Omron CX-Programmer project NewProject (CX-Programmer 9.73)

# PLC NewPLC1: CP2E-N N

## Global symbols (name address type ; comment)
0.00 BOOL  ; A/M
0.01 BOOL  ; Master On
0.03 BOOL  ; IN
0.04 BOOL  ; OUT
100.00 BOOL  ; AC 1
100.01 BOOL  ; AC 2
100.02 BOOL  ; L4
100.03 BOOL  ; L1
100.04 BOOL  ; L2
100.05 BOOL  ; L3
100.06 BOOL  ; L6
100.07 BOOL  ; L5
101.01 BOOL  ; Buzzer
10.01 BOOL  ; LAMP 4
10.02 BOOL  ; LAMP 1
10.03 BOOL  ; LAMP 2
10.04 BOOL  ; LAMP 3
10.05 BOOL  ; LAMP 6
10.06 BOOL  ; LAMP 5
1.00 BOOL  ; ON_HMI
20.00 BOOL  ; AC1
20.01 BOOL  ; LAMP 4
20.02 BOOL  ; LAMP 1
20.03 BOOL  ; LAMP 2
20.04 BOOL  ; LAMP 3
20.05 BOOL  ; LAMP 6
30.00 BOOL  ; AC 1
30.01 BOOL  ; AC 2
40.00 BOOL  ; AC 1
40.01 BOOL  ; AC 2
60.00 BOOL  ; lampu 1
60.01 BOOL  ; lampu 2
60.02 BOOL  ; lampu 3
60.03 BOOL  ; lampu 4
60.04 BOOL  ; lampu 5
60.05 BOOL  ; lampu 6
60.06 BOOL  ; AC 1
60.07 BOOL  ; AC 2
80.00 BOOL  ; AutoSet
80.01 BOOL  ; Autoful
80.02 BOOL  ; Res
90.00 BOOL  ; AUTO
90.01 BOOL  ; MANUAL
D2.00 BOOL  ; setengah
D300 CHANNEL  ; Error
D500 CHANNEL  ; ]
W60.00 BOOL  ; Setengah
Data1 D600 INT

## Program NewProgram1 (cyclic task 0)
Local symbols
Data UINT
INC BOOL
MOV BOOL
S UINT

### Section MAIN

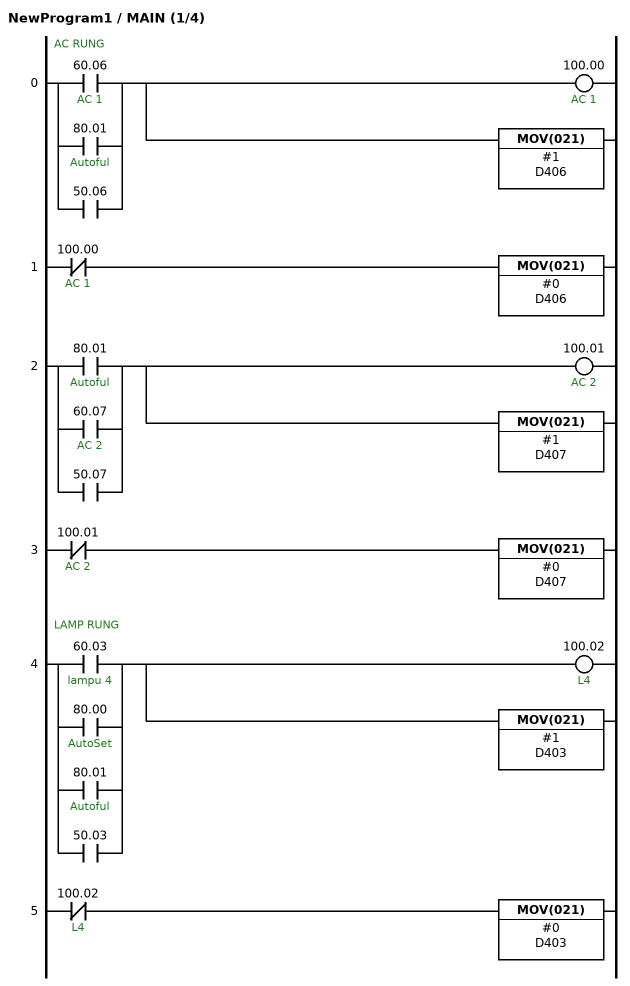
; rung 0: AC RUNG
LD 60.06  ; AC 1
OR 80.01  ; Autoful
OR 50.06
OUT 100.00  ; AC 1
MOV(021) #1 D406
; rung 1
LDNOT 100.00  ; AC 1
MOV(021) #0 D406
; rung 2
LD 80.01  ; Autoful
OR 60.07  ; AC 2
OR 50.07
OUT 100.01  ; AC 2
MOV(021) #1 D407
; rung 3
LDNOT 100.01  ; AC 2
MOV(021) #0 D407
; rung 4: LAMP RUNG
LD 60.03  ; lampu 4
OR 80.00  ; AutoSet
OR 80.01  ; Autoful
OR 50.03
OUT 100.02  ; L4
MOV(021) #1 D403
; rung 5
LDNOT 100.02  ; L4
MOV(021) #0 D403

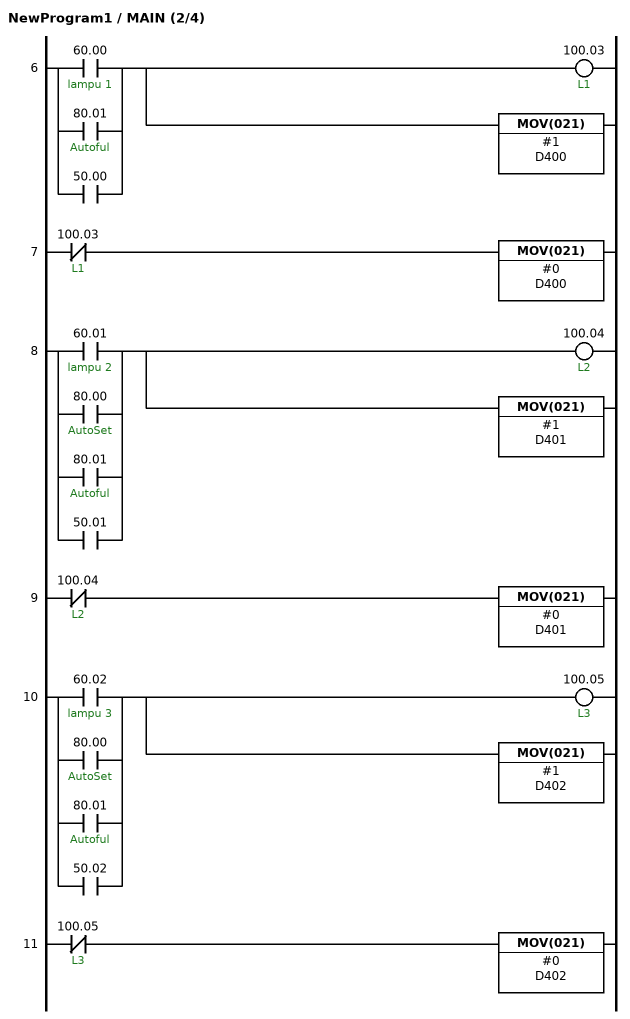
; rung 6
LD 60.00  ; lampu 1
OR 80.01  ; Autoful
OR 50.00
OUT 100.03  ; L1
MOV(021) #1 D400
; rung 7
LDNOT 100.03  ; L1
MOV(021) #0 D400
; rung 8
LD 60.01  ; lampu 2
OR 80.00  ; AutoSet
OR 80.01  ; Autoful
OR 50.01
OUT 100.04  ; L2
MOV(021) #1 D401
; rung 9
LDNOT 100.04  ; L2
MOV(021) #0 D401
; rung 10
LD 60.02  ; lampu 3
OR 80.00  ; AutoSet
OR 80.01  ; Autoful
OR 50.02
OUT 100.05  ; L3
MOV(021) #1 D402
; rung 11
LDNOT 100.05  ; L3
MOV(021) #0 D402

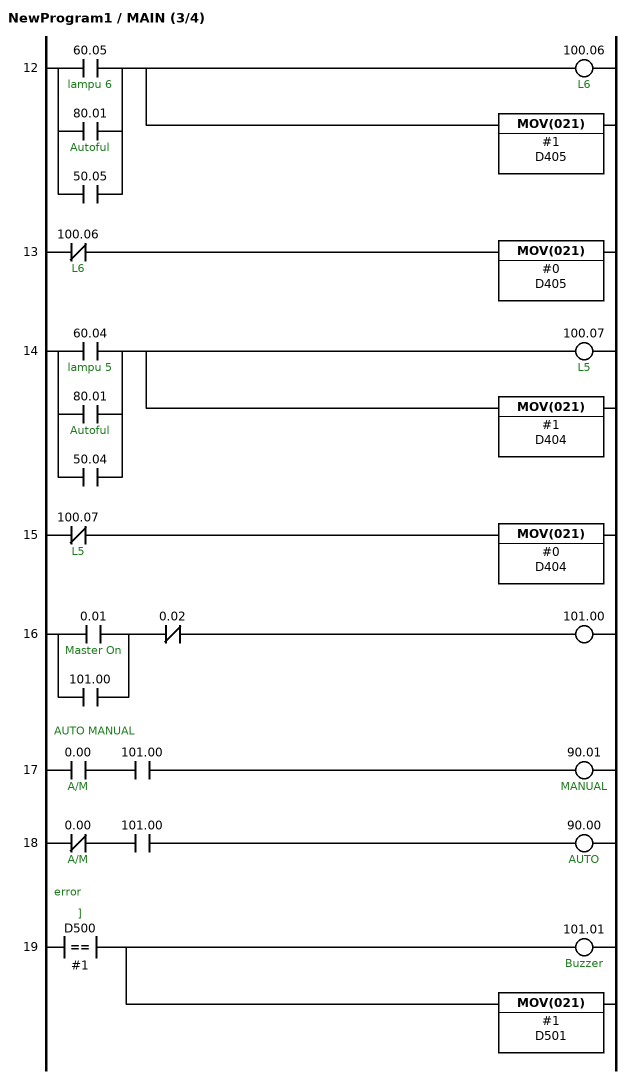
; rung 12
LD 60.05  ; lampu 6
OR 80.01  ; Autoful
OR 50.05
OUT 100.06  ; L6
MOV(021) #1 D405
; rung 13
LDNOT 100.06  ; L6
MOV(021) #0 D405
; rung 14
LD 60.04  ; lampu 5
OR 80.01  ; Autoful
OR 50.04
OUT 100.07  ; L5
MOV(021) #1 D404
; rung 15
LDNOT 100.07  ; L5
MOV(021) #0 D404
; rung 16
LD 0.01  ; Master On
OR 101.00
ANDNOT 0.02
OUT 101.00
; rung 17: AUTO MANUAL
LD 0.00  ; A/M
AND 101.00
OUT 90.01  ; MANUAL
; rung 18
LDNOT 0.00  ; A/M
AND 101.00
OUT 90.00  ; AUTO
; rung 19: error
LD=(300) D500 #1  ; ]
OUT 101.01  ; Buzzer
MOV(021) #1 D501

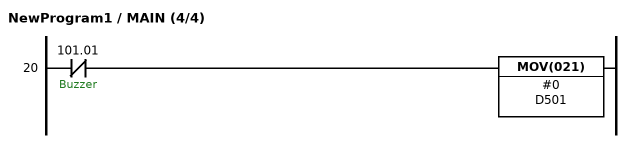
; rung 20
LDNOT 101.01  ; Buzzer
MOV(021) #0 D501

### Section MANUAL___HMI

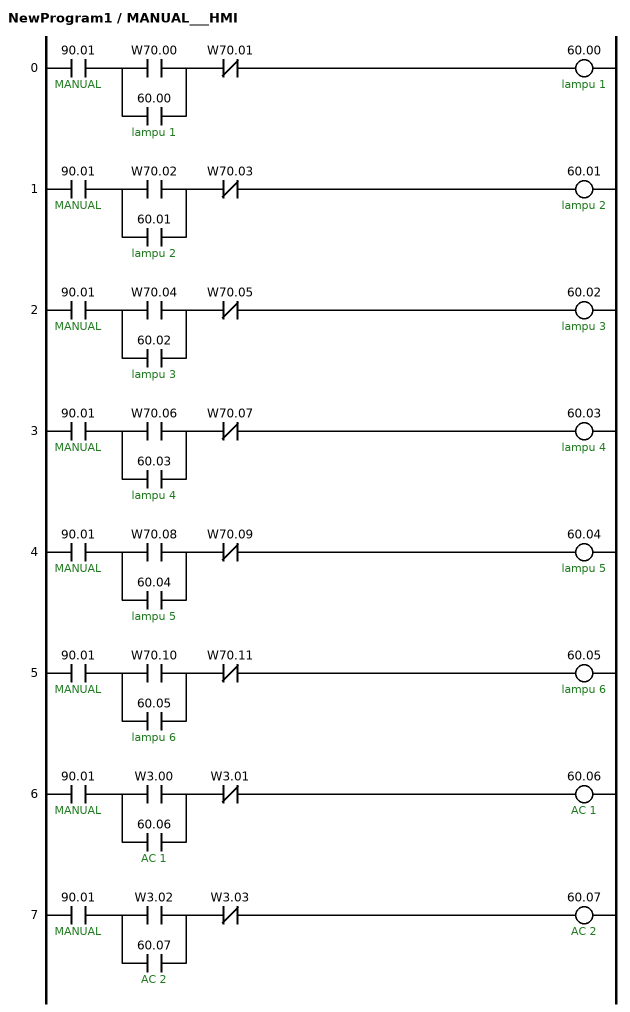
; rung 0
LD 90.01  ; MANUAL
LD W70.00
OR 60.00  ; lampu 1
ANDLD
ANDNOT W70.01
OUT 60.00  ; lampu 1
; rung 1
LD 90.01  ; MANUAL
LD W70.02
OR 60.01  ; lampu 2
ANDLD
ANDNOT W70.03
OUT 60.01  ; lampu 2
; rung 2
LD 90.01  ; MANUAL
LD W70.04
OR 60.02  ; lampu 3
ANDLD
ANDNOT W70.05
OUT 60.02  ; lampu 3
; rung 3
LD 90.01  ; MANUAL
LD W70.06
OR 60.03  ; lampu 4
ANDLD
ANDNOT W70.07
OUT 60.03  ; lampu 4
; rung 4
LD 90.01  ; MANUAL
LD W70.08
OR 60.04  ; lampu 5
ANDLD
ANDNOT W70.09
OUT 60.04  ; lampu 5
; rung 5
LD 90.01  ; MANUAL
LD W70.10
OR 60.05  ; lampu 6
ANDLD
ANDNOT W70.11
OUT 60.05  ; lampu 6
; rung 6
LD 90.01  ; MANUAL
LD W3.00
OR 60.06  ; AC 1
ANDLD
ANDNOT W3.01
OUT 60.06  ; AC 1
; rung 7
LD 90.01  ; MANUAL
LD W3.02
OR 60.07  ; AC 2
ANDLD
ANDNOT W3.03
OUT 60.07  ; AC 2

### Section AUTO

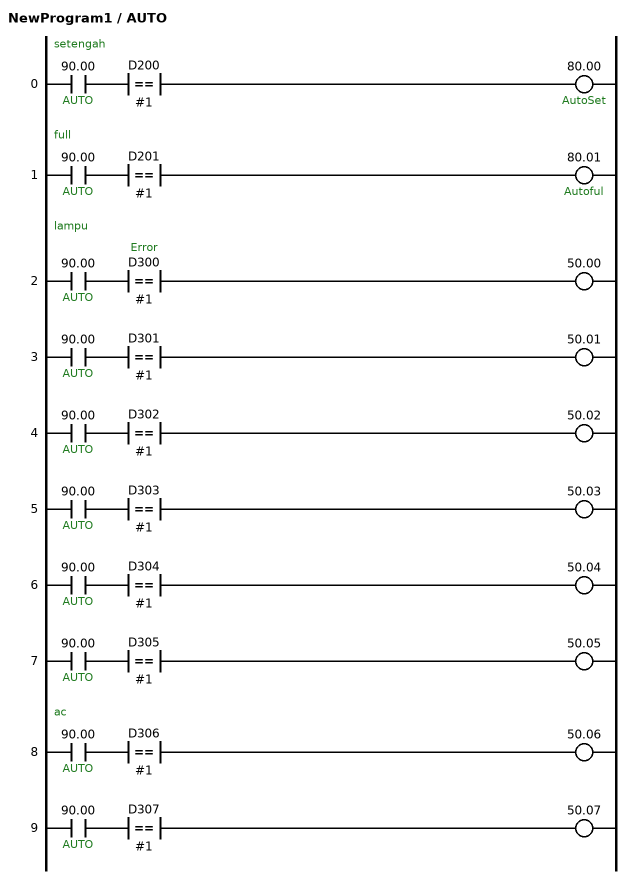
; rung 0: setengah
LD 90.00  ; AUTO
AND=(300) D200 #1
OUT 80.00  ; AutoSet
; rung 1: full
LD 90.00  ; AUTO
AND=(300) D201 #1
OUT 80.01  ; Autoful
; rung 2: lampu
LD 90.00  ; AUTO
AND=(300) D300 #1  ; Error
OUT 50.00
; rung 3
LD 90.00  ; AUTO
AND=(300) D301 #1
OUT 50.01
; rung 4
LD 90.00  ; AUTO
AND=(300) D302 #1
OUT 50.02
; rung 5
LD 90.00  ; AUTO
AND=(300) D303 #1
OUT 50.03
; rung 6
LD 90.00  ; AUTO
AND=(300) D304 #1
OUT 50.04
; rung 7
LD 90.00  ; AUTO
AND=(300) D305 #1
OUT 50.05
; rung 8: ac
LD 90.00  ; AUTO
AND=(300) D306 #1
OUT 50.06
; rung 9
LD 90.00  ; AUTO
AND=(300) D307 #1
OUT 50.07

### Section Simulator

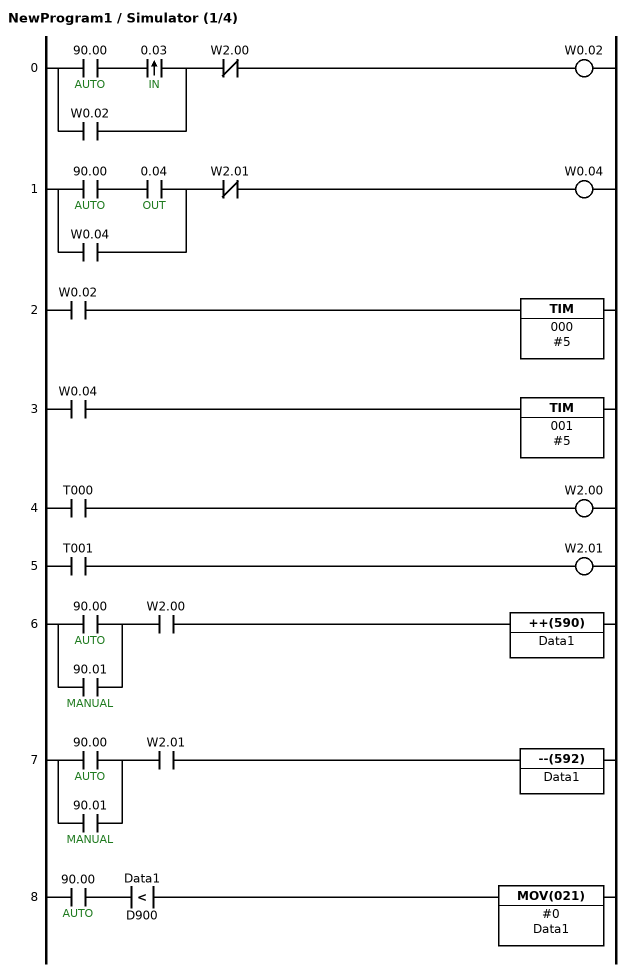
; rung 0
LD 90.00  ; AUTO
@AND 0.03  ; IN
OR W0.02
ANDNOT W2.00
OUT W0.02
; rung 1
LD 90.00  ; AUTO
AND 0.04  ; OUT
OR W0.04
ANDNOT W2.01
OUT W0.04
; rung 2
LD W0.02
TIM 000 #5
; rung 3
LD W0.04
TIM 001 #5
; rung 4
LD T000
OUT W2.00
; rung 5
LD T001
OUT W2.01
; rung 6
LD 90.00  ; AUTO
OR 90.01  ; MANUAL
AND W2.00
++(590) Data1
; rung 7
LD 90.00  ; AUTO
OR 90.01  ; MANUAL
AND W2.01
--(592) Data1
; rung 8
LD 90.00  ; AUTO
AND<S(312) Data1 D900
MOV(021) #0 Data1

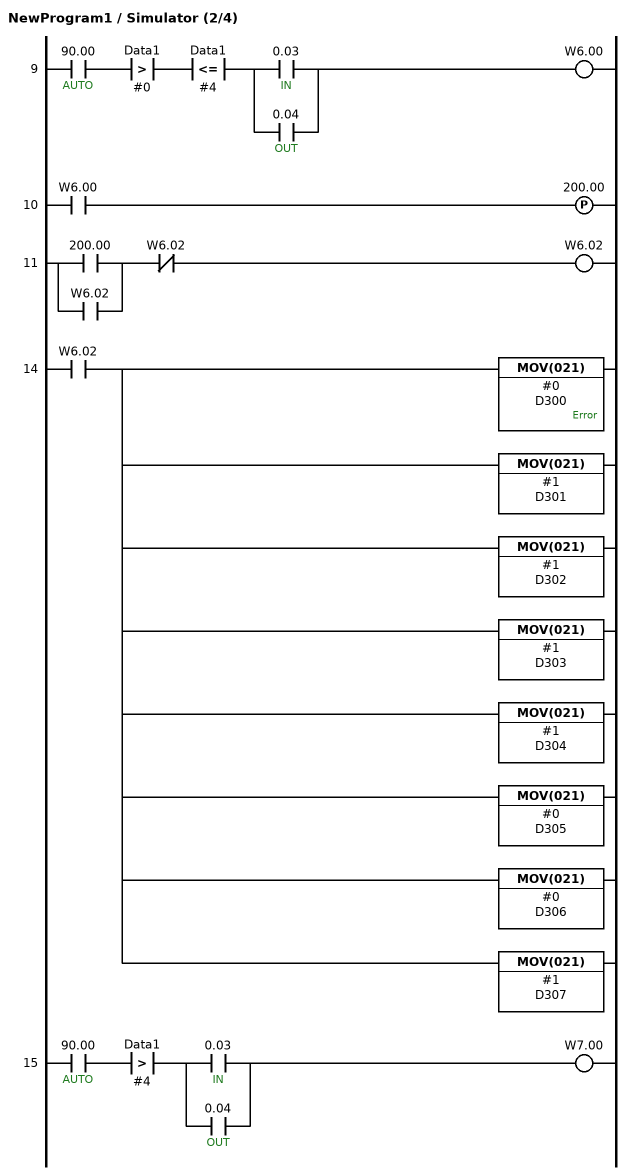
; rung 9
LD 90.00  ; AUTO
AND>S(322) Data1 #0
AND<=(315) Data1 #4
LD 0.03  ; IN
OR 0.04  ; OUT
ANDLD
OUT W6.00
; rung 10
LD W6.00
DIFU(013) 200.00
; rung 11
LD 200.00
OR W6.02
ANDNOT W6.02
OUT W6.02
; rung 14
LD W6.02
MOV(021) #0 D300  ; Error
MOV(021) #1 D301
MOV(021) #1 D302
MOV(021) #1 D303
MOV(021) #1 D304
MOV(021) #0 D305
MOV(021) #0 D306
MOV(021) #1 D307
; rung 15
LD 90.00  ; AUTO
AND>S(322) Data1 #4
LD 0.03  ; IN
OR 0.04  ; OUT
ANDLD
OUT W7.00

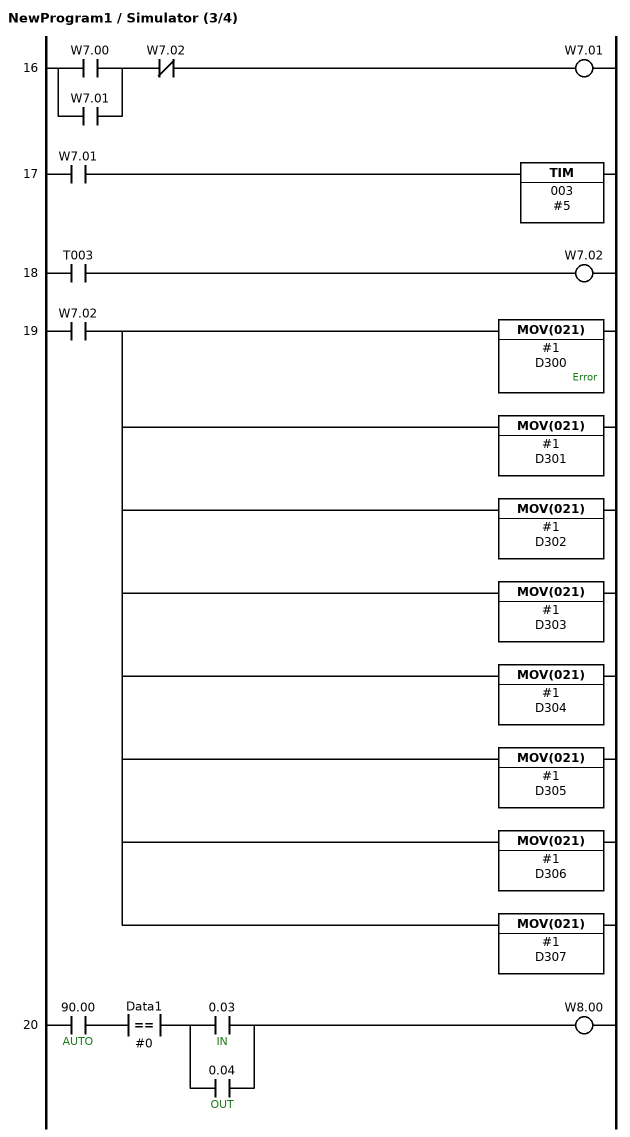
; rung 16
LD W7.00
OR W7.01
ANDNOT W7.02
OUT W7.01
; rung 17
LD W7.01
TIM 003 #5
; rung 18
LD T003
OUT W7.02
; rung 19
LD W7.02
MOV(021) #1 D300  ; Error
MOV(021) #1 D301
MOV(021) #1 D302
MOV(021) #1 D303
MOV(021) #1 D304
MOV(021) #1 D305
MOV(021) #1 D306
MOV(021) #1 D307
; rung 20
LD 90.00  ; AUTO
AND=S(302) Data1 #0
LD 0.03  ; IN
OR 0.04  ; OUT
ANDLD
OUT W8.00

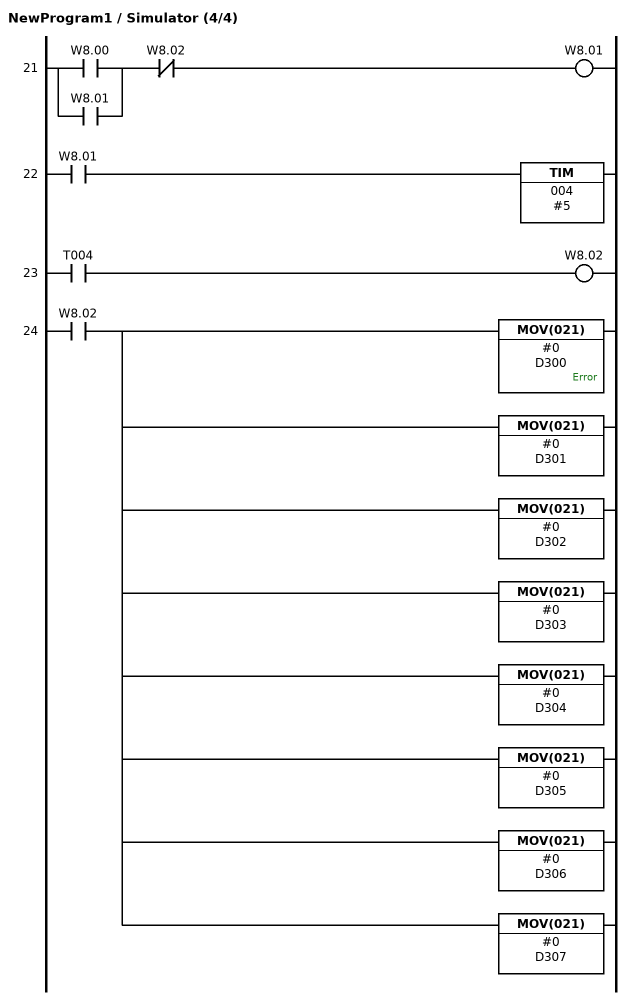
; rung 21
LD W8.00
OR W8.01
ANDNOT W8.02
OUT W8.01
; rung 22
LD W8.01
TIM 004 #5
; rung 23
LD T004
OUT W8.02
; rung 24
LD W8.02
MOV(021) #0 D300  ; Error
MOV(021) #0 D301
MOV(021) #0 D302
MOV(021) #0 D303
MOV(021) #0 D304
MOV(021) #0 D305
MOV(021) #0 D306
MOV(021) #0 D307

### Section END
; rung 0
END(001)